// TIA Portal V15.1 export
// export: Created 2020-06-12T07:35:38.4287109Z, ExportSetting None, DisplayName Totally Integrated Automation Portal, DisplayVersion V15.1, DisplayName TIA Portal Openness, DisplayVersion V15.1, DisplayName STEP 7 Professional, DisplayVersion V15.1, DisplayName STEP 7 Safety, DisplayVersion V15.1, DisplayName WinCC Advanced, DisplayVersion V15.1
FUNCTION "F_export" : Void   // FC53, F_FBD
TITLE = Export F-data to user DB
{ S7_Optimized_Access := 'TRUE' }
BEGIN

REGION Network 1: Inputs ES1GD01 keys
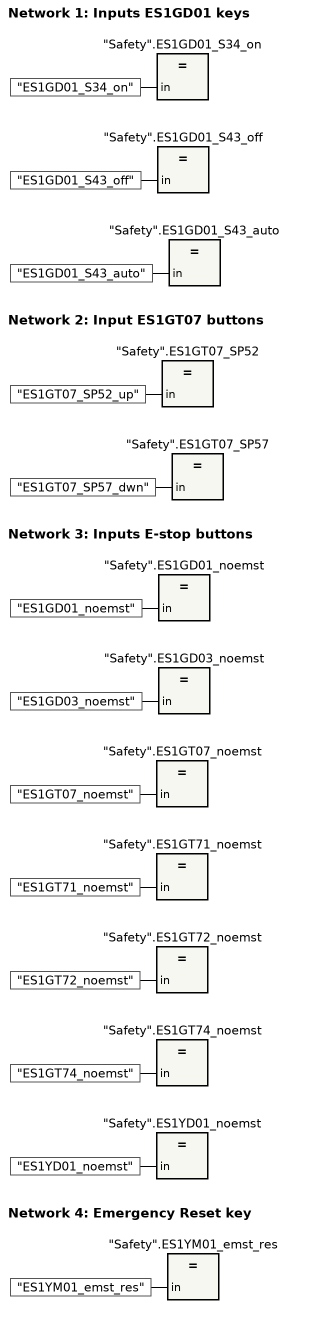
   "Safety".ES1GD01_S34_on := "ES1GD01_S34_on";
   "Safety".ES1GD01_S43_off := "ES1GD01_S43_off";
   "Safety".ES1GD01_S43_auto := "ES1GD01_S43_auto";
END_REGION

REGION Network 2: Input ES1GT07 buttons
   "Safety".ES1GT07_SP52 := "ES1GT07_SP52_up";
   "Safety".ES1GT07_SP57 := "ES1GT07_SP57_dwn";
END_REGION

REGION Network 3: Inputs E-stop buttons
   "Safety".ES1GD01_noemst := "ES1GD01_noemst";
   "Safety".ES1GD03_noemst := "ES1GD03_noemst";
   "Safety".ES1GT07_noemst := "ES1GT07_noemst";
   "Safety".ES1GT71_noemst := "ES1GT71_noemst";
   "Safety".ES1GT72_noemst := "ES1GT72_noemst";
   "Safety".ES1GT74_noemst := "ES1GT74_noemst";
   "Safety".ES1YD01_noemst := "ES1YD01_noemst";
END_REGION

REGION Network 4: Emergency Reset key
   "Safety".ES1YM01_emst_res := "ES1YM01_emst_res";
END_REGION

REGION Network 5: Limit / Door / Ladder / Safety switches
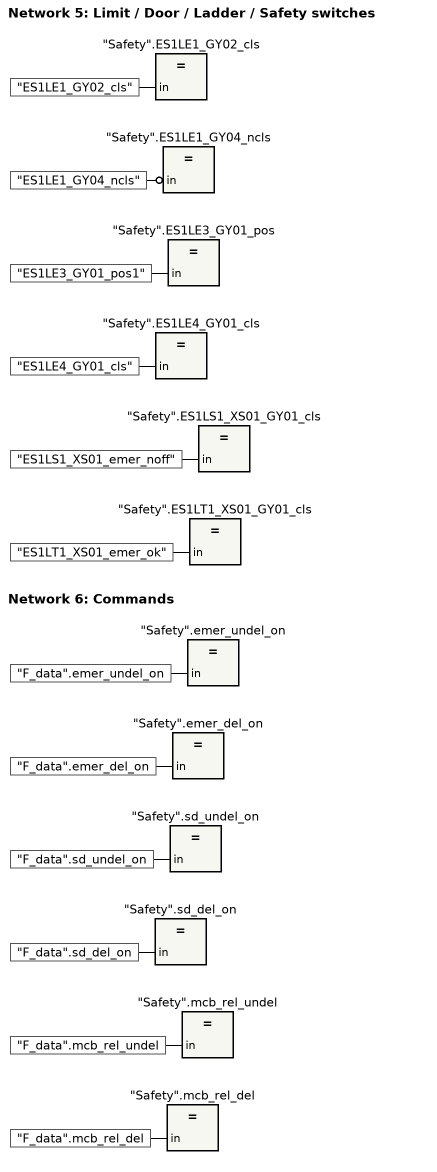
   "Safety".ES1LE1_GY02_cls := "ES1LE1_GY02_cls";
   "Safety".ES1LE1_GY04_ncls := NOT "ES1LE1_GY04_ncls";
   "Safety".ES1LE3_GY01_pos := "ES1LE3_GY01_pos1";
   "Safety".ES1LE4_GY01_cls := "ES1LE4_GY01_cls";
   "Safety".ES1LS1_XS01_GY01_cls := "ES1LS1_XS01_emer_noff";
   "Safety".ES1LT1_XS01_GY01_cls := "ES1LT1_XS01_emer_ok";
END_REGION

REGION Network 6: Commands
   "Safety".emer_undel_on := "F_data".emer_undel_on;
   "Safety".emer_del_on := "F_data".emer_del_on;
   "Safety".sd_undel_on := "F_data".sd_undel_on;
   "Safety".sd_del_on := "F_data".sd_del_on;
   "Safety".mcb_rel_undel := "F_data".mcb_rel_undel;
   "Safety".mcb_rel_del := "F_data".mcb_rel_del;
END_REGION

REGION Network 7: Emergency line outputs
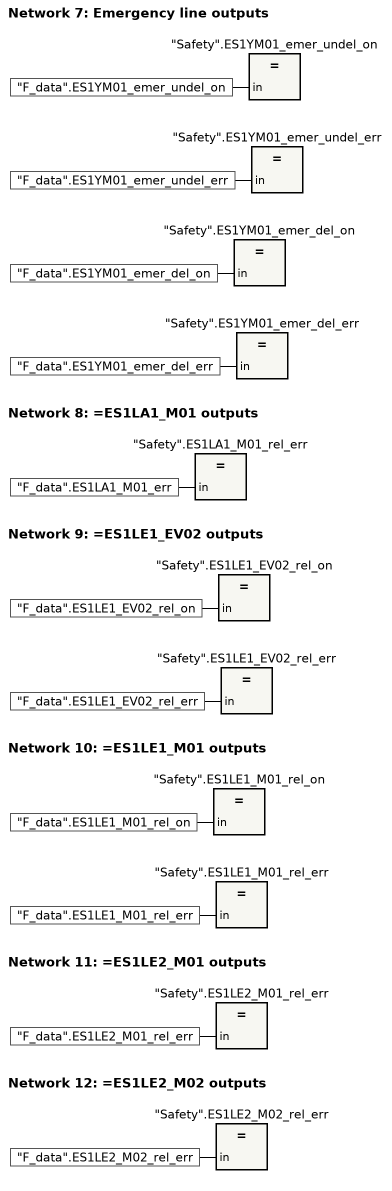
   "Safety".ES1YM01_emer_undel_on := "F_data".ES1YM01_emer_undel_on;
   "Safety".ES1YM01_emer_undel_err := "F_data".ES1YM01_emer_undel_err;
   "Safety".ES1YM01_emer_del_on := "F_data".ES1YM01_emer_del_on;
   "Safety".ES1YM01_emer_del_err := "F_data".ES1YM01_emer_del_err;
END_REGION

REGION Network 8: =ES1LA1_M01 outputs
   "Safety".ES1LA1_M01_rel_err := "F_data".ES1LA1_M01_err;
END_REGION

REGION Network 9: =ES1LE1_EV02 outputs
   "Safety".ES1LE1_EV02_rel_on := "F_data".ES1LE1_EV02_rel_on;
   "Safety".ES1LE1_EV02_rel_err := "F_data".ES1LE1_EV02_rel_err;
END_REGION

REGION Network 10: =ES1LE1_M01 outputs
   "Safety".ES1LE1_M01_rel_on := "F_data".ES1LE1_M01_rel_on;
   "Safety".ES1LE1_M01_rel_err := "F_data".ES1LE1_M01_rel_err;
END_REGION

REGION Network 11: =ES1LE2_M01 outputs
   "Safety".ES1LE2_M01_rel_err := "F_data".ES1LE2_M01_rel_err;
END_REGION

REGION Network 12: =ES1LE2_M02 outputs
   "Safety".ES1LE2_M02_rel_err := "F_data".ES1LE2_M02_rel_err;
END_REGION

REGION Network 13: =ES1LE3_M01 outputs
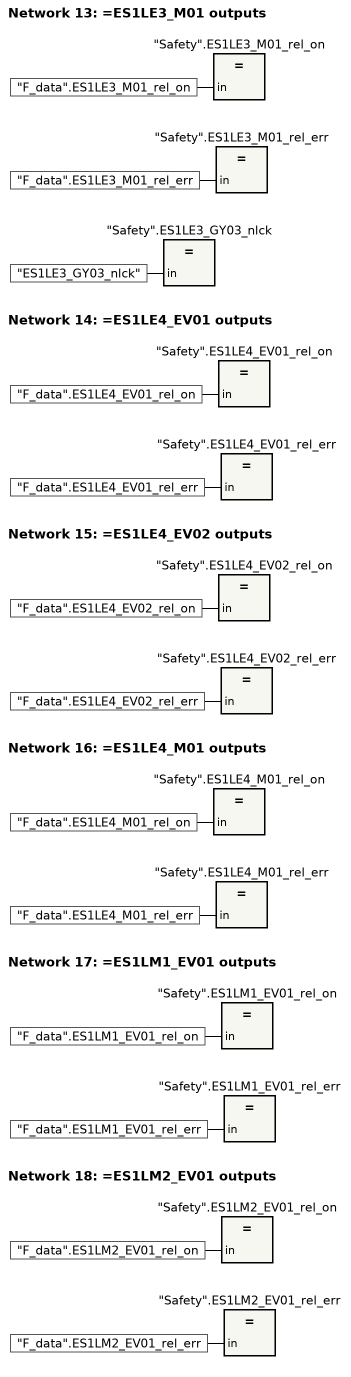
   "Safety".ES1LE3_M01_rel_on := "F_data".ES1LE3_M01_rel_on;
   "Safety".ES1LE3_M01_rel_err := "F_data".ES1LE3_M01_rel_err;
   "Safety".ES1LE3_GY03_nlck := "ES1LE3_GY03_nlck";
END_REGION

REGION Network 14: =ES1LE4_EV01 outputs
   "Safety".ES1LE4_EV01_rel_on := "F_data".ES1LE4_EV01_rel_on;
   "Safety".ES1LE4_EV01_rel_err := "F_data".ES1LE4_EV01_rel_err;
END_REGION

REGION Network 15: =ES1LE4_EV02 outputs
   "Safety".ES1LE4_EV02_rel_on := "F_data".ES1LE4_EV02_rel_on;
   "Safety".ES1LE4_EV02_rel_err := "F_data".ES1LE4_EV02_rel_err;
END_REGION

REGION Network 16: =ES1LE4_M01 outputs
   "Safety".ES1LE4_M01_rel_on := "F_data".ES1LE4_M01_rel_on;
   "Safety".ES1LE4_M01_rel_err := "F_data".ES1LE4_M01_rel_err;
END_REGION

REGION Network 17: =ES1LM1_EV01 outputs
   "Safety".ES1LM1_EV01_rel_on := "F_data".ES1LM1_EV01_rel_on;
   "Safety".ES1LM1_EV01_rel_err := "F_data".ES1LM1_EV01_rel_err;
END_REGION

REGION Network 18: =ES1LM2_EV01 outputs
   "Safety".ES1LM2_EV01_rel_on := "F_data".ES1LM2_EV01_rel_on;
   "Safety".ES1LM2_EV01_rel_err := "F_data".ES1LM2_EV01_rel_err;
END_REGION

REGION Network 19: =ES1LS1_XS01 outputs
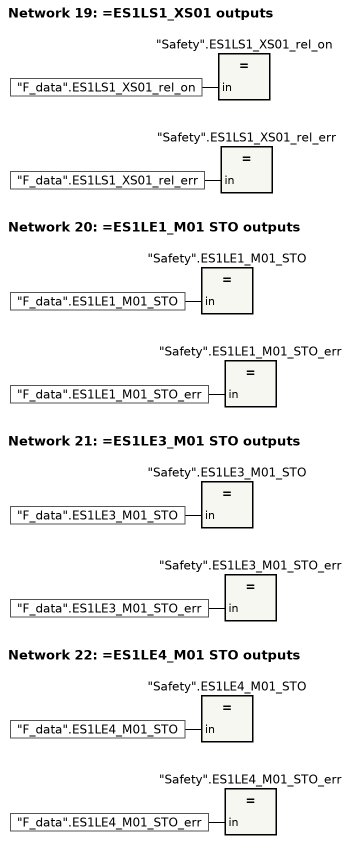
   "Safety".ES1LS1_XS01_rel_on := "F_data".ES1LS1_XS01_rel_on;
   "Safety".ES1LS1_XS01_rel_err := "F_data".ES1LS1_XS01_rel_err;
END_REGION

REGION Network 20: =ES1LE1_M01 STO outputs
   "Safety".ES1LE1_M01_STO := "F_data".ES1LE1_M01_STO;
   "Safety".ES1LE1_M01_STO_err := "F_data".ES1LE1_M01_STO_err;
END_REGION

REGION Network 21: =ES1LE3_M01 STO outputs
   "Safety".ES1LE3_M01_STO := "F_data".ES1LE3_M01_STO;
   "Safety".ES1LE3_M01_STO_err := "F_data".ES1LE3_M01_STO_err;
END_REGION

REGION Network 22: =ES1LE4_M01 STO outputs
   "Safety".ES1LE4_M01_STO := "F_data".ES1LE4_M01_STO;
   "Safety".ES1LE4_M01_STO_err := "F_data".ES1LE4_M01_STO_err;
END_REGION

REGION Network 23: !!!!!!!!!!!!!!!!!!!!!!!!!!!!!!!!!!!!!!!!!!!!!!!!!!!!!!!!!!!!!!!!!!!!!!!! Delete me Simulator !!!!!!!!!!!!!!!!!!!!!!!!!!!!!!!!!!!!!!!!!!!!!!
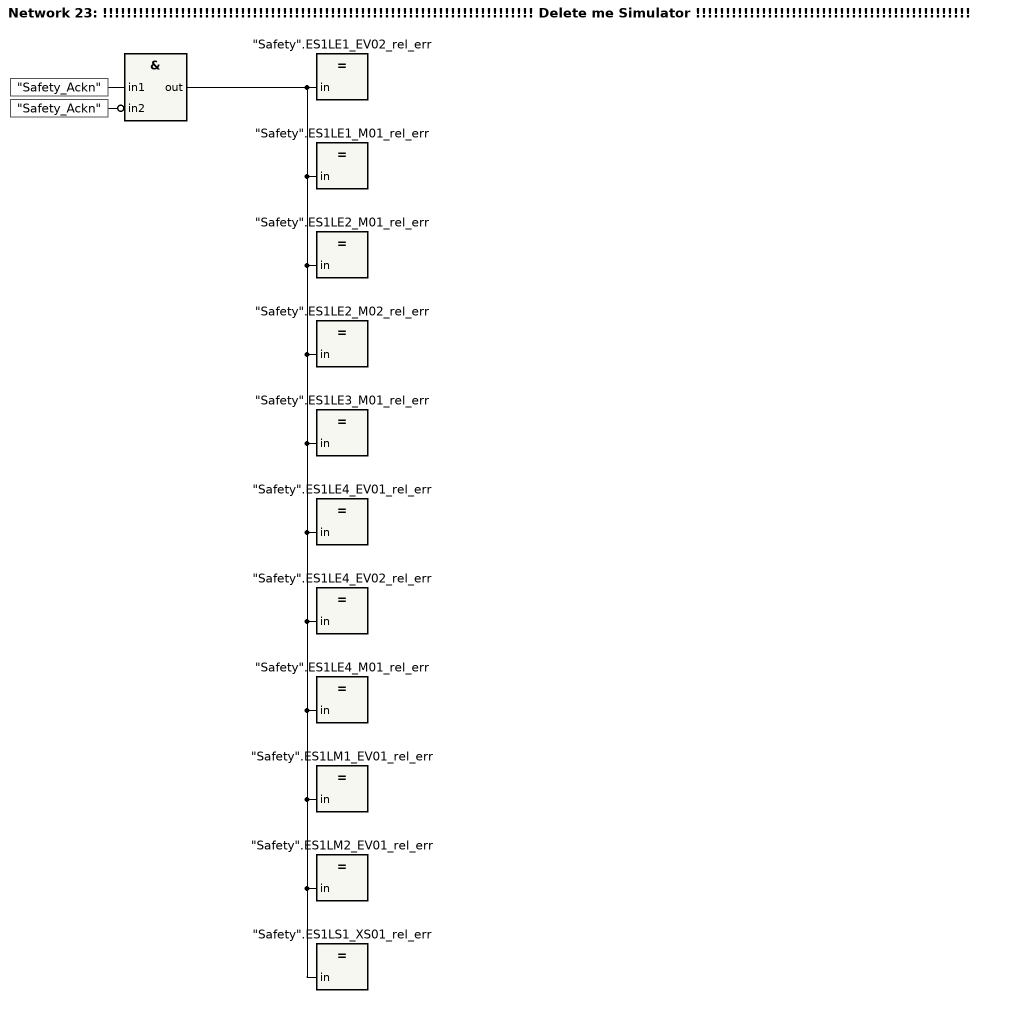
   "Safety".ES1LE1_EV02_rel_err := "Safety_Ackn" AND NOT "Safety_Ackn";
   "Safety".ES1LE1_M01_rel_err := "Safety".ES1LE1_EV02_rel_err;
   "Safety".ES1LE2_M01_rel_err := "Safety".ES1LE1_EV02_rel_err;
   "Safety".ES1LE2_M02_rel_err := "Safety".ES1LE1_EV02_rel_err;
   "Safety".ES1LE3_M01_rel_err := "Safety".ES1LE1_EV02_rel_err;
   "Safety".ES1LE4_EV01_rel_err := "Safety".ES1LE1_EV02_rel_err;
   "Safety".ES1LE4_EV02_rel_err := "Safety".ES1LE1_EV02_rel_err;
   "Safety".ES1LE4_M01_rel_err := "Safety".ES1LE1_EV02_rel_err;
   "Safety".ES1LM1_EV01_rel_err := "Safety".ES1LE1_EV02_rel_err;
   "Safety".ES1LM2_EV01_rel_err := "Safety".ES1LE1_EV02_rel_err;
   "Safety".ES1LS1_XS01_rel_err := "Safety".ES1LE1_EV02_rel_err;
END_REGION

REGION Network 24: !!!!!!!!!!!!!!!!!!!!!!!!!!!!!!!!!!!!!!!!!!!!!!!!!!!!!!!!!!!!!!!!!!!!!!!! Delete me Simulator !!!!!!!!!!!!!!!!!!!!!!!!!!!!!!!!!!!!!!!!!!!!!!
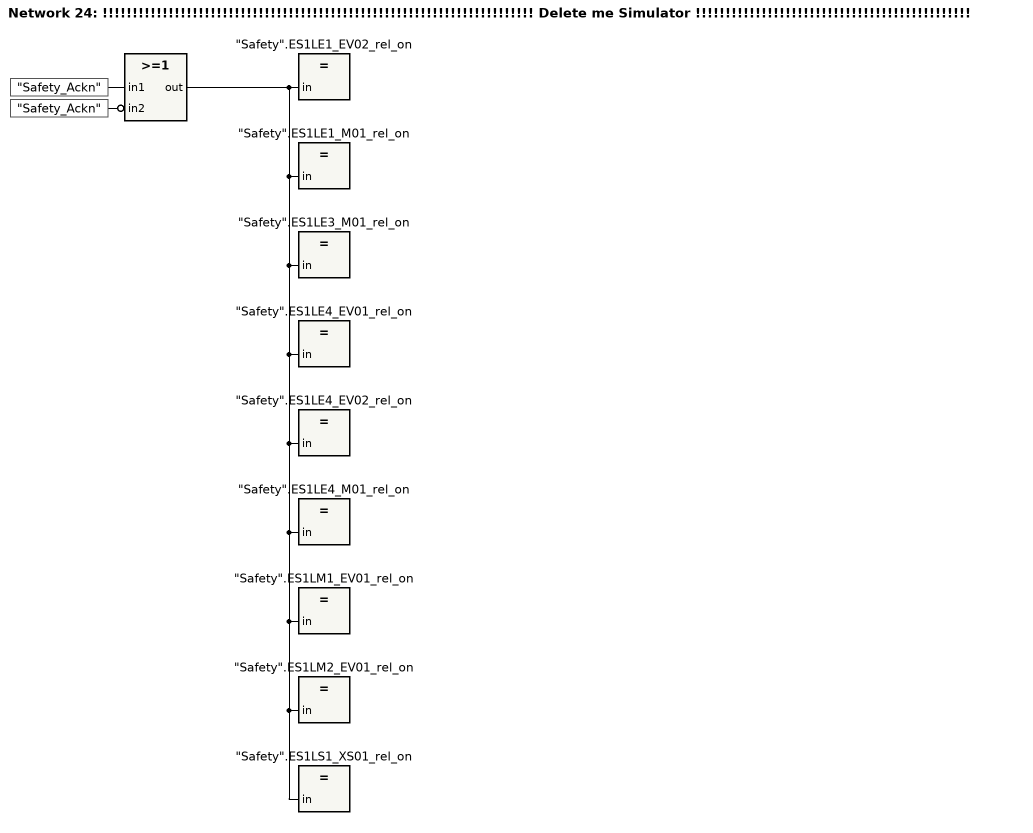
   "Safety".ES1LE1_EV02_rel_on := "Safety_Ackn" OR NOT "Safety_Ackn";
   "Safety".ES1LE1_M01_rel_on := "Safety".ES1LE1_EV02_rel_on;
   "Safety".ES1LE3_M01_rel_on := "Safety".ES1LE1_EV02_rel_on;
   "Safety".ES1LE4_EV01_rel_on := "Safety".ES1LE1_EV02_rel_on;
   "Safety".ES1LE4_EV02_rel_on := "Safety".ES1LE1_EV02_rel_on;
   "Safety".ES1LE4_M01_rel_on := "Safety".ES1LE1_EV02_rel_on;
   "Safety".ES1LM1_EV01_rel_on := "Safety".ES1LE1_EV02_rel_on;
   "Safety".ES1LM2_EV01_rel_on := "Safety".ES1LE1_EV02_rel_on;
   "Safety".ES1LS1_XS01_rel_on := "Safety".ES1LE1_EV02_rel_on;
END_REGION
END_FUNCTION
